KUKA KRL program: chk_w6_grp2_opn.src

&ACCESS RVO1
&COMMENT Accelo Z2.1_Z2.2
DEF chk_w6_grp2_opn( )
; Check gripper ACCELO OPEN Z2.1 Z2.2
;//---- Start User-------

$TIMER[10] = 0
$TIMER_STOP[10] = FALSE

WAIT FOR ($IN[37] AND $IN[39] AND $IN[41])
WAIT FOR (NOT $IN[38] AND NOT $IN[40] AND NOT $IN[42])

$TIMER_STOP[10] = TRUE
$TIMER[10] = 0

;//---- End User---------
END
